FUNCTION_BLOCK GetInstancePath (* Service Interface Function Block Type *)
  PACKAGE eclipse4diac::utils;
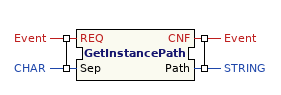
  EVENT_INPUT
    REQ WITH Sep; (* Service Request *)
  END_EVENT
  EVENT_OUTPUT
    CNF WITH Path; (* Confirmation of Requested Service *)
  END_EVENT
  VAR_INPUT
    Sep : CHAR := '/'; (* Separator character for the output path generated by this FB *)
  END_VAR
  VAR_OUTPUT
    Path : STRING; (* Instance path of this FB *)
  END_VAR
  SERVICE APPLICATION/RESOURCE (* Service Interface Function Block Type *)
    SEQUENCE Normal_Operation
      APPLICATION.REQ(Sep) -> RESOURCE.acquire path information(Sep) -> APPLICATION.CNF(Path);
    END_SEQUENCE
  END_SERVICE
END_FUNCTION_BLOCK
